PROGRAM P_Inputs
VAR
	fbJoystickLeftVert 					: FB_JoystickInputScaling;
	fbJoystickLeftHor 					: FB_JoystickInputScaling;
	
	fbJoystickRightVert 				: FB_JoystickInputScaling;
	fbJoystickRightHor 					: FB_JoystickInputScaling;
	
	bEnableJoystick : BOOL;
		
END_VAR

bEnableJoystick := NOT(P_StablePlatform.bManualMode);

fbJoystickLeftVert(
	bEnable := bEnableJoystick,
	nRawInput := G_Inputs.stJoyLY.nValue,
	stJoystickInputScaling := G_Parameters.stParam.stJoystickInputScalingLeftY,
	fNormalizedOutput => G_Sensors.fJoystickLeftNormalizedY
);

IF G_Sensors.fJoystickLeftNormalizedY < 0 THEN
	G_Sensors.MCDirectionAxis3 := MC_Negative_Direction;
ELSIF G_Sensors.fJoystickLeftNormalizedY > 0 THEN
	G_Sensors.MCDirectionAxis3 := MC_Positive_Direction;	
END_IF

fbJoystickLeftHor(
	bEnable := bEnableJoystick,
	nRawInput := G_Inputs.stJoyLX.nValue,
	stJoystickInputScaling := G_Parameters.stParam.stJoystickInputScalingLeftX,
	fNormalizedOutput => G_Sensors.fJoystickLeftNormalizedX
);

IF G_Sensors.fJoystickLeftNormalizedX < 0 THEN
	G_Sensors.MCDirectionAxis1 := MC_Positive_Direction;
ELSIF G_Sensors.fJoystickLeftNormalizedX > 0 THEN
	G_Sensors.MCDirectionAxis1 := MC_Negative_Direction;	
END_IF


fbJoystickRightVert(
	bEnable := bEnableJoystick,
	nRawInput := G_Inputs.stJoyRY.nValue,
	stJoystickInputScaling := G_Parameters.stParam.stJoystickInputScalingRightY,
	fNormalizedOutput => G_Sensors.fJoystickRightNormalizedY
);

IF G_Sensors.fJoystickRightNormalizedY < 0 THEN
	G_Sensors.MCDirectionAxis4 := MC_Negative_Direction;
ELSIF G_Sensors.fJoystickRightNormalizedY > 0 THEN
	G_Sensors.MCDirectionAxis4 := MC_Positive_Direction;	
END_IF



fbJoystickRightHor(
	bEnable := bEnableJoystick,
	nRawInput := G_Inputs.stJoyRX.nValue,
	stJoystickInputScaling := G_Parameters.stParam.stJoystickInputScalingRightX,
	fNormalizedOutput => G_Sensors.fJoystickRightNormalizedX
);

IF G_Sensors.fJoystickRightNormalizedX < 0 THEN
	G_Sensors.MCDirectionAxis2 := MC_Positive_Direction;
ELSIF G_Sensors.fJoystickRightNormalizedX > 0 THEN
	G_Sensors.MCDirectionAxis2 := MC_Negative_Direction;	
END_IF

END_PROGRAM

(* stored: Version 1.1.0.1, ProductVersion 3.1.4024.12
   POU P_Inputs: Id {8b676dbd-393f-42d6-8803-330b6e90ab14}, SpecialFunc None *)
